PROGRAM MAIN
VAR
	AngleDeg : LREAL;
	AngleRad : LREAL;
END_VAR

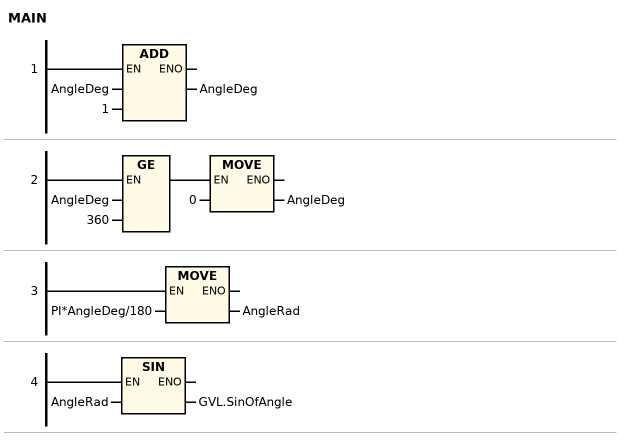
// NETWORK 1
AngleDeg := AngleDeg + 1;

// NETWORK 2
IF AngleDeg >= 360 THEN AngleDeg := 0; END_IF

// NETWORK 3
AngleRad := PI*AngleDeg/180;

// NETWORK 4
GVL.SinOfAngle := SIN(AngleRad);

END_PROGRAM

(* stored: Version 1.1.0.1, ProductVersion 3.1.4024.12
   POU MAIN: Id {49e7dad4-0d20-4f11-9de4-71670c409dd2}, SpecialFunc None *)
